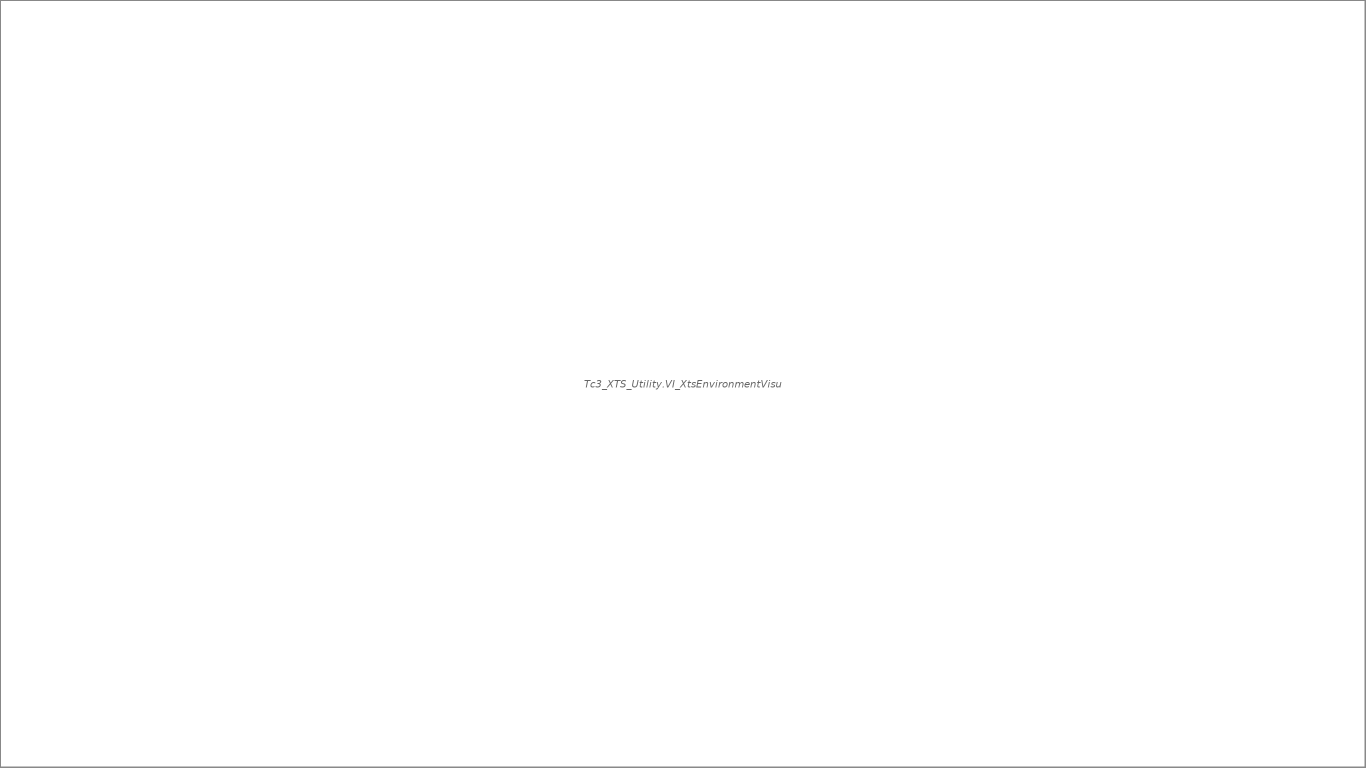
VISUALIZATION DiagnosticVisu  // 1366x768
    Frame (0,0 1366x768)
        shows Tc3_XTS_Utility.VI_XtsEnvironmentVisu()
END_VISUALIZATION

(* stored: Version 1.1.0.1, ProductVersion 3.1.4026.12
   Visu DiagnosticVisu: Id {31b0087d-1c58-4879-b1c9-5319ad10b809} *)
